Staubli VAL3: HerePoint.pgx

public program HerePoint(num x_nIndex)
  local tool l_tTool
  local point l_pHere
  local frame l_fFrame
  local num i
  local num l_nIndex
begin
  //
  // take the point
  //
  jEditPoint.tData[x_nIndex].jJoint=herej()
  resetMotion()
end
